// TwinCAT 3 PLC project TankFillingSystem
// ProgramVersion: 3.1.4024.0
// libraries:
//   Tc2_Standard, * (Beckhoff Automation GmbH)
//   Tc2_System, * (Beckhoff Automation GmbH)
//   Tc3_Module, * (Beckhoff Automation GmbH)
// project tree:
//   / PlcTask.TcTTO
//   POUs/ FB_AdjustablePump.TcPOU, FB_Controller.TcPOU, FB_FixedPump.TcPOU, I_AdjustablePump.TcIO, I_Pump.TcIO, MAIN.TcPOU
// (motion and I/O tree: see PLC project functionblockpractice)
// real-time tasks:
//   TASK PlcTask: cycle T#10ms, priority 20, ADS port 350
//   TASK PlcTask2: cycle T#10ms, priority 22, ADS port 352
//   TASK PlcTask1: cycle T#10ms, priority 21, ADS port 351
//   TASK PlcTask3: cycle T#10ms, priority 23, ADS port 353

CONFIGURATION TankFillingSystem
    RESOURCE PLC ON TwinCAT3
        TASK PlcTask(INTERVAL := T#10ms, PRIORITY := 23);
        PROGRAM MAIN WITH PlcTask : MAIN;
    END_RESOURCE
END_CONFIGURATION

// ---- POUs/I_AdjustablePump.TcIO
INTERFACE I_AdjustablePump EXTENDS I_Pump, __SYSTEM.IQueryInterface

METHOD SetFlowRate : BOOL
VAR_INPUT
	fNewRate : REAL;
END_VAR
END_METHOD

END_INTERFACE

// ---- POUs/I_Pump.TcIO
INTERFACE I_Pump EXTENDS __SYSTEM.IQueryInterface

METHOD GetFlowRate : REAL
VAR_INPUT
END_VAR
END_METHOD

METHOD GetTotalVolume : REAL
VAR_INPUT
END_VAR
END_METHOD

METHOD Start : BOOL
VAR_INPUT
END_VAR
END_METHOD

METHOD Stop : BOOL
VAR_INPUT
END_VAR
END_METHOD

END_INTERFACE

// ---- POUs/MAIN.TcPOU
PROGRAM MAIN
VAR
	fbFixedPump1 : FB_FixedPump;
	fbAdjustPump2 : FB_AdjustablePump;
	
	fbController1 : FB_Controller(fbFixedPump1);
	fbController2 : FB_Controller(fbAdjustPump2);
	
	fNewRate : REAL := 40;
	
	bOn : BOOL;
	bOff : BOOL;
	
END_VAR

IF bOn THEN
	fbController1.bPumpOn := TRUE;
	fbController1.fNewRate := fNewRate;
	fbController2.bPumpOn := TRUE;
	fbController2.fNewRate := fNewRate;
END_IF
IF bOff THEN
	fbController1.bPumpOn := FALSE;
	fbController2.bPumpOn := FALSE;
	fbController1.bPumpOff := TRUE;
	fbController2.bPumpOff := TRUE;
END_IF


fbFixedPump1();
fbAdjustPump2();
fbController1();
fbController2();

END_PROGRAM

// ---- POUs/FB_FixedPump.TcPOU
FUNCTION_BLOCK FB_FixedPump IMPLEMENTS I_Pump


VAR CONSTANT
	fFlowRate : REAL := 20 ;
END_VAR
VAR
	bRunning : BOOL;
	fTotalVolume : REAL;
END_VAR

IF bRunning THEN
	fTotalVolume := fTotalVolume + fFlowRate;
END_IF

{warning 'add method implementation '}
METHOD GetFlowRate : REAL
GetFlowRate := fFlowRate;
END_METHOD

{warning 'add method implementation '}
METHOD GetTotalVolume : REAL
GetTotalVolume := fTotalVolume;
END_METHOD

{warning 'add method implementation '}
METHOD Start : BOOL
Start := bRunning := TRUE;
END_METHOD

{warning 'add method implementation '}
METHOD Stop : BOOL
bRunning := FALSE;
Stop := TRUE;
END_METHOD

END_FUNCTION_BLOCK

// ---- POUs/FB_AdjustablePump.TcPOU
FUNCTION_BLOCK FB_AdjustablePump IMPLEMENTS I_AdjustablePump

VAR
	bRunning : BOOL;
	fTotalVolume : REAL;
	fFlowRate : REAL := 20;
END_VAR

IF bRunning THEN
	fTotalVolume := fTotalVolume + fFlowRate;
END_IF

{warning 'add method implementation '}
METHOD GetFlowRate : REAL
GetFlowRate := fFlowRate;
END_METHOD

{warning 'add method implementation '}
METHOD GetTotalVolume : REAL
GetTotalVolume := fTotalVolume;
END_METHOD

METHOD SetFlowRate : BOOL
VAR_INPUT
	fNewRate : REAL;
END_VAR
fFlowRate := fNewRate;
END_METHOD

{warning 'add method implementation '}
METHOD Start : BOOL
Start := bRunning := TRUE;
END_METHOD

{warning 'add method implementation '}
METHOD Stop : BOOL
bRunning := FALSE;
END_METHOD

END_FUNCTION_BLOCK

// ---- POUs/FB_Controller.TcPOU
FUNCTION_BLOCK FB_Controller
VAR_INPUT
	fNewRate : REAL;
	bPumpOn : BOOL;
	bPumpOff : BOOL;
END_VAR
VAR
	iPump : I_Pump;
	iAdjustPump : I_AdjustablePump;
	bAdjustable : BOOL;
END_VAR

IF bPumpOn THEN
	IF iPump <> 0 THEN
		iPump.Start();
		IsAdjustable();
		IF bAdjustable THEN
		iAdjustPump.SetFlowRate(fNewRate);
		END_IF
	END_IF
END_IF
IF bPumpOff THEN
	IF iPump <> 0 THEN
		iPump.Stop();
	END_IF
	
END_IF

METHOD FB_init : BOOL
VAR_INPUT
	bInitRetains : BOOL; // if TRUE, the retain variables are initialized (warm start / cold start)
	bInCopyCode : BOOL;  // if TRUE, the instance afterwards gets moved into the copy code (online change)
	_iPump : I_Pump;
END_VAR
iPump := _iPump;
END_METHOD

METHOD IsAdjustable 
VAR_INPUT
END_VAR
bAdjustable := __QUERYINTERFACE(iPump, iAdjustPump);
END_METHOD

END_FUNCTION_BLOCK
